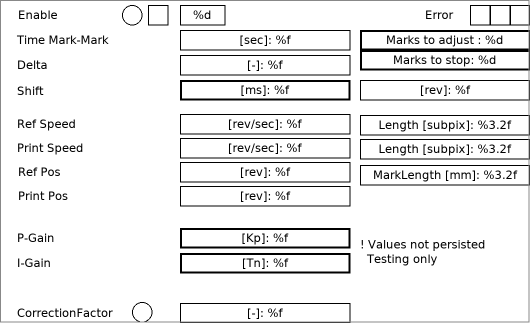
VISUALIZATION _VISU_DRIFTCONTROL  // 530x323
VAR_IN_OUT
  mRef  : FB_DRIFTCONTROL;
END_VAR
    Rectangle (15,5 97x20), "Enable"
    RoundedRectangle (148,5 20x20), colour toggle: mRef.bL_ControlActive
    Ellipse (122,5 20x20), colour toggle: mRef.bI_Enable
        toggle mRef.bI_Enable
    Rectangle (14,30 120x20), "Time Mark-Mark"
    Rectangle (180,30 170x20), "[sec]: %f", text variable: mRef.fL_DeltaTimeStamp
    Rectangle (14,55 120x20), "Delta"
    Rectangle (180,55 170x20), "[-]: %f", text variable: mRef.fL_DeltaCtrl
    Rectangle (14,228 120x20), "P-Gain"
    Rectangle (180,228 170x20), "[Kp]: %f", text variable: mRef.fI_ControllerPGain
        OnMouseDown: write the text variable via Default
    Rectangle (14,253 120x20), "I-Gain"
    Rectangle (180,253 170x20), "[Tn]: %f", text variable: mRef.fI_ControllerIGain
        OnMouseDown: write the text variable via Edit
    Rectangle (14,303 120x20), "CorrectionFactor"
    Rectangle (180,303 170x20), "[-]: %f", text variable: mRef.fO_SpeedCorrectionFactor
    Rectangle (14,114 120x20), "Ref Speed"
    Rectangle (180,114 170x20), "[rev/sec]: %f", text variable: mRef.fL_RefSpeed
    Rectangle (14,138 120x20), "Print Speed"
    Rectangle (180,138 170x20), "[rev/sec]: %f", text variable: mRef.fL_ImgSpeed
    Ellipse (132,302 20x20), colour toggle: mRef.bI_OutputEnable
        toggle mRef.bI_OutputEnable
    Rectangle (360,115 170x20), "Length [subpix]: %3.2f", text variable: mRef.fL_RefLength, colour toggle: mRef.bL_FormatWarning
    Rectangle (360,139 170x20), "Length [subpix]: %3.2f", text variable: mRef.lL_ImgLength, colour toggle: mRef.bL_FormatWarning
    Rectangle (15,162 120x20), "Ref Pos"
    Rectangle (180,162 170x20), "[rev]: %f", text variable: mRef.fL_RefPos
    Rectangle (15,186 120x20), "Print Pos"
    Rectangle (180,186 170x20), "[rev]: %f", text variable: mRef.fL_ImgPos
    RoundedRectangle (470,5 20x20), tooltip "ctrl err", colour toggle: mRef.bO_ContrErr
        tap mRef.bL_ResetInternal
    Rectangle (422,5 42x20), "Error"
    Rectangle (357,233 141x38), "! Values not persisted Testing only"
    Rectangle (180,80 170x20), "[ms]: %f", text variable: mRef.fI_DriftTimeShift
        OnMouseDown: write the text variable via Default
    Rectangle (14,81 120x20), "Shift"
    Rectangle (360,80 170x20), "[rev]: %f", text variable: mRef.fL_ShiftPos
    Rectangle (180,5 45x20), "%d", text variable: mRef.iL_State
    RoundedRectangle (490,5 20x20), tooltip "fb err", colour toggle: mRef.bL_Error
        tap mRef.bL_ResetInternal
    RoundedRectangle (510,5 20x20), tooltip "arw", colour toggle: mRef.fL_CtrlGainFactor <> 1
        tap mRef.bL_ResetInternal
    Rectangle (360,165 170x20), "MarkLength [mm]: %3.2f", text variable: mRef.fL_RefLengthMM, colour toggle: mRef.bL_FormatWarning
    Rectangle (360,30 170x20), "Marks to adjust : %d", text variable: mRef.nI_NbCyclesToAdjust, colour toggle: mRef.bO_ControllerAdjusted
        OnMouseDown: write the text variable via Default
    Rectangle (360,50 170x20), "Marks to stop: %d", text variable: mRef.nI_NbMissMarksToStop, colour toggle: mRef.bO_ControllerAdjusted
        OnMouseDown: write the text variable via Default
END_VISUALIZATION

(* stored: Version 1.1.0.1, ProductVersion 3.1.4024.11
   Visu _VISU_DRIFTCONTROL: Id {54d8ba90-325f-43de-847e-cf544b8af54b} *)
